// TIA Portal project "Soru1" (V15)

(* hardware
DEVICE "S7-1200 station_1"  S7-1200 Station
   slot 0: "Rack_0"  S7-1200 Rack  Rack  V1.0
   slot 1: "PLC_1"  CPU 1214C DC/DC/DC  6ES7 214-1AG40-0XB0  V4.2
*)

// ===== PLC "PLC_1"  CPU 1214C DC/DC/DC =====

VAR_GLOBAL   // PLC tag table "Default tag table"
   "Stop" AT %I0.0 : Bool;
   "Start" AT %I0.1 : Bool;
   "AA1" AT %I0.2 : Bool;
   "AA2" AT %I0.3 : Bool;
   "Motor_1" AT %Q0.0 : Bool;
   "Motor_2" AT %Q0.1 : Bool;
END_VAR

// folder: System blocks/Program resources

DATA_BLOCK "zaman"   // DB1
{ S7_Optimized_Access := 'TRUE' }
AUTHOR : Simatic
FAMILY : IEC
NAME : IEC_TMR
VERSION : 1.0
// stored: InstanceOfName IEC_TIMER
"IEC_TIMER"
BEGIN
END_DATA_BLOCK

// folder: (top level)

ORGANIZATION_BLOCK "Main"   // OB1, LAD, ProgramCycle
TITLE = "Main Program Sweep (Cycle)"
{ S7_Optimized_Access := 'TRUE' }
VERSION : 0.1
   VAR_INPUT
      Initial_Call : Bool;   // Initial call of this OB
      Remanence : Bool;   // =True, if remanent data are available
   END_VAR
BEGIN

REGION Network 1
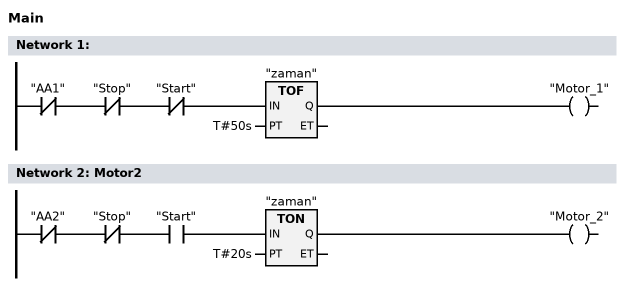
   "zaman".TOF(IN := NOT "AA1" AND NOT "Stop" AND NOT "Start", PT := T#50s);
   "Motor_1" := "zaman".Q;
END_REGION

REGION Network 2: Motor2
   "zaman".TON(IN := NOT "AA2" AND NOT "Stop" AND "Start", PT := T#20s);
   "Motor_2" := "zaman".Q;
END_REGION
END_ORGANIZATION_BLOCK